// TIA Portal V21 export
DATA_BLOCK "ComunicazioneS7_St1_Qci"   // DB9000
{ S7_Optimized_Access := 'FALSE' }
   VAR
      Recive : Struct
         Watchdog_Bit : Bool := TRUE;   // WATCH DOG (LIFE BIT)
         BOOL_SIGNAL_2 : Bool := TRUE;
         BOOL_SIGNAL_3 : Bool := FALSE;
         BOOL_SIGNAL_4 : Bool := FALSE;
         BOOL_SIGNAL_5 : Bool := TRUE;
         BOOL_SIGNAL_6 : Bool := FALSE;
         BOOL_SIGNAL_7 : Bool := FALSE;
         BOOL_SIGNAL_8 : Bool := FALSE;
         BOOL_SIGNAL_9 : Bool := FALSE;
         BOOL_SIGNAL_10 : Bool := FALSE;
         BOOL_SIGNAL_11 : Bool := FALSE;
         BOOL_SIGNAL_12 : Bool := FALSE;
         BOOL_SIGNAL_13 : Bool := FALSE;
         BOOL_SIGNAL_14 : Bool := FALSE;
         BOOL_SIGNAL_15 : Bool := FALSE;
         BOOL_SIGNAL_16 : Bool := FALSE;
         BOOL_SIGNAL_17 : Bool := FALSE;
         BOOL_SIGNAL_18 : Bool := FALSE;
         BOOL_SIGNAL_19 : Bool := FALSE;
         BOOL_SIGNAL_20 : Bool := FALSE;
         BOOL_SIGNAL_21 : Bool := FALSE;
         BOOL_SIGNAL_22 : Bool := FALSE;
         BOOL_SIGNAL_23 : Bool := FALSE;
         BOOL_SIGNAL_24 : Bool := FALSE;
         Watchdog_Incrementale : DInt := 0;
         DINT_SIGNAL_2 : DInt := 0;
         DINT_SIGNAL_3 : DInt := 0;
         DINT_SIGNAL_4 : DInt := 0;
         DINT_SIGNAL_5 : DInt := 0;
         DINT_SIGNAL_6 : DInt := 0;
         DINT_SIGNAL_7 : DInt := 0;
         DINT_SIGNAL_8 : DInt := 0;
         DINT_SIGNAL_9 : DInt := 0;
         DINT_SIGNAL_10 : DInt := 0;
         DINT_SIGNAL_11 : DInt := 0;
         DINT_SIGNAL_12 : DInt := 0;
         DINT_SIGNAL_13 : DInt := 0;
         DINT_SIGNAL_14 : DInt := 0;
         DINT_SIGNAL_15 : DInt := 0;
         DINT_SIGNAL_16 : DInt := 0;
         DINT_SIGNAL_17 : DInt := 0;
         DINT_SIGNAL_18 : DInt := 0;
         DINT_SIGNAL_19 : DInt := 0;
         DINT_SIGNAL_20 : DInt := 0;
         REAL_SIGNAL_1 : Real := 0.0;
         REAL_SIGNAL_2 : Real := 0.0;
         REAL_SIGNAL_3 : Real := 0.0;
         REAL_SIGNAL_4 : Real := 80.0;
         REAL_SIGNAL_5 : Real := 80.0;
         REAL_SIGNAL_6 : Real := 0.0;
         REAL_SIGNAL_7 : Real := 0.0;
         REAL_SIGNAL_8 : Real := 0.0;
         REAL_SIGNAL_9 : Real := 0.0;
         REAL_SIGNAL_10 : Real := 0.0;
         REAL_SIGNAL_11 : Real := 0.0;
         REAL_SIGNAL_12 : Real := 0.0;
         REAL_SIGNAL_13 : Real := 0.0;
         REAL_SIGNAL_14 : Real := 0.0;
         REAL_SIGNAL_15 : Real := 0.0;
         REAL_SIGNAL_16 : Real := 0.0;
         REAL_SIGNAL_17 : Real := 0.0;
         REAL_SIGNAL_18 : Real := 0.0;
         REAL_SIGNAL_19 : Real := 0.0;
         REAL_SIGNAL_20 : Real := 0.0;
      END_STRUCT;
      Send : Struct
         Watchdog_Bit : Bool := TRUE;   // WATCH DOG (LIFE BIT)
         ChiamataProdotto : Bool := TRUE;   // Chiamata prodotto
         BOOL_SIGNAL_3 : Bool := TRUE;
         BOOL_SIGNAL_4 : Bool := FALSE;
         BOOL_SIGNAL_5 : Bool := FALSE;
         BOOL_SIGNAL_6 : Bool := FALSE;
         BOOL_SIGNAL_7 : Bool := FALSE;
         BOOL_SIGNAL_8 : Bool := FALSE;
         BOOL_SIGNAL_9 : Bool := FALSE;
         BOOL_SIGNAL_10 : Bool := FALSE;
         BOOL_SIGNAL_11 : Bool := FALSE;
         BOOL_SIGNAL_12 : Bool := FALSE;
         BOOL_SIGNAL_13 : Bool := FALSE;
         BOOL_SIGNAL_14 : Bool := FALSE;
         BOOL_SIGNAL_15 : Bool := FALSE;
         BOOL_SIGNAL_16 : Bool := FALSE;
         BOOL_SIGNAL_17 : Bool := FALSE;
         BOOL_SIGNAL_18 : Bool := FALSE;
         BOOL_SIGNAL_19 : Bool := FALSE;
         BOOL_SIGNAL_20 : Bool := FALSE;
         BOOL_SIGNAL_21 : Bool := FALSE;
         BOOL_SIGNAL_22 : Bool := FALSE;
         BOOL_SIGNAL_23 : Bool := FALSE;
         BOOL_SIGNAL_24 : Bool := FALSE;
         Watchdog_Incrementale : DInt := 0;
         DINT_SIGNAL_2 : DInt := 0;
         DINT_SIGNAL_3 : DInt := 0;
         DINT_SIGNAL_4 : DInt := 0;
         DINT_SIGNAL_5 : DInt := 0;
         DINT_SIGNAL_6 : DInt := 0;
         DINT_SIGNAL_7 : DInt := 0;
         DINT_SIGNAL_8 : DInt := 0;
         DINT_SIGNAL_9 : DInt := 0;
         DINT_SIGNAL_10 : DInt := 0;
         DINT_SIGNAL_11 : DInt := 0;
         DINT_SIGNAL_12 : DInt := 0;
         DINT_SIGNAL_13 : DInt := 0;
         DINT_SIGNAL_14 : DInt := 0;
         DINT_SIGNAL_15 : DInt := 0;
         DINT_SIGNAL_16 : DInt := 0;
         DINT_SIGNAL_17 : DInt := 0;
         DINT_SIGNAL_18 : DInt := 0;
         DINT_SIGNAL_19 : DInt := 0;
         DINT_SIGNAL_20 : DInt := 0;
         LivelloAttualeSerbatoio : Real := 69.85083;   // Livello attuale serbatoio prodotto
         REAL_SIGNAL_2 : Real := 0.0;
         REAL_SIGNAL_3 : Real := 0.0;
         REAL_SIGNAL_4 : Real := 0.0;
         REAL_SIGNAL_5 : Real := 0.0;
         REAL_SIGNAL_6 : Real := 0.0;
         REAL_SIGNAL_7 : Real := 0.0;
         REAL_SIGNAL_8 : Real := 0.0;
         REAL_SIGNAL_9 : Real := 0.0;
         REAL_SIGNAL_10 : Real := 0.0;
         REAL_SIGNAL_11 : Real := 0.0;
         REAL_SIGNAL_12 : Real := 0.0;
         REAL_SIGNAL_13 : Real := 0.0;
         REAL_SIGNAL_14 : Real := 0.0;
         REAL_SIGNAL_15 : Real := 0.0;
         REAL_SIGNAL_16 : Real := 0.0;
         REAL_SIGNAL_17 : Real := 0.0;
         REAL_SIGNAL_18 : Real := 0.0;
         REAL_SIGNAL_19 : Real := 0.0;
         REAL_SIGNAL_20 : Real := 0.0;
      END_STRUCT;
   END_VAR
BEGIN
END_DATA_BLOCK
